// TwinCAT 3 PLC project Hausaufgaben
// ProgramVersion: 3.1.4026.16
// libraries:
//   Tc2_Standard, * (Beckhoff Automation GmbH)
//   Tc2_System, * (Beckhoff Automation GmbH)
// project tree:
//   / PlcTask.TcTTO (not stored)
//   POUs/ FlipFlopR1.TcPOU (not stored), FlipFlopS1.TcPOU, MAIN.TcPOU, RSFlipFlop.TcPOU (not stored), ScaleFB.TcPOU (not stored), SRFlipFlop.TcPOU
// real-time tasks:
//   TASK PlcTask: cycle T#10ms, priority 20, ADS port 350
//   TASK PlcTask1: cycle T#10ms, priority 21, ADS port 351

// ---- POUs/FlipFlopS1.TcPOU
FUNCTION_BLOCK FlipFlopS1
VAR_INPUT							//S-Dominanter FlipFlop mit negiertem Reseteingang
	bSET: BOOL;						//Baustein-interne Set-Variable
	bRESET: BOOL;					//Baustein-interne Reset-Variable
END_VAR
VAR_OUTPUT
	bQ1: BOOL;						//Baustein-interne Ausgangs-Variable
END_VAR
VAR
END_VAR

IF bSET								//Abfrage ob Set = 1, da S-Dominant 
	THEN
	bQ1 := TRUE;
ELSIF NOT bRESET AND NOT bSET 		//Abfrage ob Reset = 0 und nicht Set = 1
	THEN
	bQ1 := FALSE;
END_IF

END_FUNCTION_BLOCK

// ---- POUs/MAIN.TcPOU
PROGRAM MAIN
VAR
	FlipFlopRS_Baustein: RSFlipFlop;	// Instanzierung des RS-Bibliothek-Bausteins
	FlipFlopSR_Baustein: SRFlipFlop;	// Instanzierung des SR-Bibliothek-Bausteins
	SR: FlipFlopR1;						// Instanzierung des SR-Bausteins mit IF, ELSIF
	RS: FlipFlopS1;						// Instanzierung des RS-Bausteins mit IF, ELSIF
    Ix_TasterOn: BOOL;  				// Set-Eingang
    Ix_TasterOff: BOOL; 				// Reset-Eingang
    bQRS: BOOL;							// RS-Ausgang mit IF, ELSIF
	bQSR: BOOL;							// SR-Ausgang mit IF, ELSIF
	bQRSBaustein: BOOL;					// RS-Ausgang mit Bibliothek-Baustein
	bQSRBaustein: BOOL;					// SR-Ausgang mit Bibliothek-Baustein
	iSensor: INT;						// Eingang Analogsensor 
	iScaledValue: INT;					// Skalierter Wert des Analogsensors
	ScaleFB: ScaleFB;					// Instanzierung des Scale-Bausteins
	END_VAR

// RS(bSET := Ix_TasterOn, bRESET := Ix_TasterOff);					//Aufruf des RS-Bausteins + Verknüpfung der I/Os (IF, ELSIF)
// bQRS := RS.bQ1;														//Zuweisung des entsprechenden Ausgangs
// 
// SR(bSET := Ix_TasterOn, bRESET := Ix_TasterOff);					//Aufruf des SR-Bausteins + Verknüpfung der I/Os (IF, ELSIF)
// bQSR := SR.bQ1;														//Zuweisung des entsprechenden Ausgangs
// 
// FlipFlopRS_Baustein(bSET:= Ix_TasterOn, bRESET:= NOT Ix_TasterOff);	//Aufruf des RS-Bausteines + Verknüpfung der I/Os, mit RS-Baustein aus der Bibliothek
// bQRSBaustein:= RS.bQ1;												//Zuweisung des entsprechenden Ausgangs
// 			
// FlipFlopSR_Baustein(bSET:= Ix_TasterOn, bRESET:= Ix_TasterOff);		//Aufruf des SR-Bausteines + Verknüpfung der I/Os, mit SR-Baustein aus der Bibliothek
// bQSRBaustein:= SR.bQ1;												//Zuweisung des entsprechenden Ausgangs

// ScaleFB(iRohWert:= iSensor);
// iScaledValue:= ScaleFB.ScaledValue;

END_PROGRAM

// ---- POUs/SRFlipFlop.TcPOU
FUNCTION_BLOCK SRFlipFlop
VAR_INPUT										//R-Dominanter RS-Baustein
	bSET: BOOL;									//Baustein-interne Set-Variable
	bRESET: BOOL;								//Baustein-interne Reset-Variable
END_VAR
VAR_OUTPUT
END_VAR
VAR
	SRFlipFlop: SR;								//Instanziierung des SR-Bausteins
END_VAR

SRFlipFlop(SET1:= bSET, RESET:= bRESET);		//Verknüpfung der Baustein-internen Variablen mit den Bausteineingängen

END_FUNCTION_BLOCK
